TYPE TcoUr20_Outputs_v_1_x_x :
STRUCT
	Outputs AT %Q* : ARRAY[0..63] OF BYTE;
END_STRUCT
END_TYPE

(* stored: Version 1.1.0.1, ProductVersion 3.1.4024.12
   DUT TcoUr20_Outputs_v_1_x_x: Id {3c55fecb-0b12-0baf-2e2b-4b75d91af754} *)
